TYPE "MEStoPLC_AlarmMassage_ext"
VERSION : 0.1
   STRUCT
      ErrorCode : Int;
      StatusBits : DInt;
      Cycle_ID : DInt;
      Unit_ParttypeID : Int;
      "Transfer time" : String[60];
   END_STRUCT;

END_TYPE

